PROGRAM _3000_PRG_Running
VAR_IN_OUT
    CurrentStep : ActiveStep;  // Shared step structure with state machine
	NextStep: DINT; // Next step to be modified by sequences
END_VAR
VAR_INPUT
    StepTimerSeconds : DINT;   // Timer value from state machine
    RetrySignal : BOOL;        // Retry signal from state machine
    StateMachineStatus : ST_SM_Status;  // Complete state machine status
END_VAR

VAR
    // Step function blocks for running sequence
    fbStep3000 : FB_SequenceStep;  // Production Start
    fbStep3002 : FB_SequenceStep;  // Production Execute
    fbStep3004 : FB_SequenceStep;  // Production Quality Check
    fbStep3006 : FB_SequenceStep;  // Packaging Prepare
    fbStep3008 : FB_SequenceStep;  // Production Finalize
    
    // Step permissives (simulation for testing)
    step3000Perms : INT := -1;     // All OK for step 3000
    step3002Perms : INT := -1;     // All OK for step 3002
    step3004Perms : INT := -1;     // All OK for step 3004
    step3006Perms : INT := -1;     // All OK for step 3006
    step3008Perms : INT := -1;     // All OK for step 3008
    
END_VAR

//=============================================================================
// PRG_Running - Handles RUNNING state sequence (3000-3999)
//=============================================================================
// Step numbering: 3000, 3002 (even numbers)
// Fault steps: 3001, 3003 (odd numbers, +1 of original)
// NOTE: Initial step setting (CurrentStep.Step = 0) is handled in MAIN program


//=============================================================================
// STEP 3000 - PRODUCTION START
//=============================================================================
fbStep3000(
    inpStep := CurrentStep.Step,
    cfgStep := 3000,
    cfgNextStep := 3002,
    inpStepTimerSeconds := StepTimerSeconds,
    inpRetry := RetrySignal,
    inpStepPermissives := step3000Perms,
    cfgStepTimeout := 12,  // 12 second timeout
    inpFaultStep := FALSE,
    ActiveStep := CurrentStep
);

// Step 3000 Active Logic
IF fbStep3000.outStepActive THEN
    // Only simulate permissives if step is active but not advancing
    IF fbStep3000.outNextStep = fbStep3000.cfgStep THEN  // Step is waiting for permissives
        // Permissives simulation - Simulate based on timer
        IF StepTimerSeconds < 5 THEN
            step3000Perms := 16#FFFE;  // Bit 0 not OK (not ready yet)
        ELSE
            step3000Perms := -1;  // All permissives OK after 5 seconds
        END_IF;
    END_IF;
    
    // HMI configuration and actions
    CurrentStep.PermsHMI.Name := 'Production Start';
    CurrentStep.PermsHMI.Desc[0] := 'Raw Material Available';
    CurrentStep.PermsHMI.Desc[1] := 'Process Temperature OK';
    CurrentStep.PermsHMI.Desc[2] := 'Quality System Ready';
    
    // Add any step-specific actions here
    // Example: Start production line, initialize process parameters, etc.
    
    // FB_SequenceStep determines next step automatically based on permissives
    NextStep := fbStep3000.outNextStep;
ELSE
    // Reset permissives when step is not active (ensures fresh start next time)
    step3000Perms := 16#FFFE;  // Reset to NOT OK when leaving step
END_IF;

//=============================================================================
// STEP 3002 - PRODUCTION EXECUTE
//=============================================================================
fbStep3002(
    inpStep := CurrentStep.Step,
    cfgStep := 3002,
    cfgNextStep := 3004,
    inpStepTimerSeconds := StepTimerSeconds,
    inpRetry := RetrySignal,
    inpStepPermissives := step3002Perms,
    cfgStepTimeout := 20,  // 20 second timeout
    inpFaultStep := FALSE,
    ActiveStep := CurrentStep
);

// Step 3002 Active Logic
IF fbStep3002.outStepActive THEN
    // Only simulate permissives if step is active but not advancing
    IF fbStep3002.outNextStep = fbStep3002.cfgStep THEN  // Step is waiting for permissives
        // Permissives simulation - Simulate based on timer
        IF StepTimerSeconds < 15 THEN
            step3002Perms := 16#FFFD;  // Bit 1 not OK (production not complete)
        ELSE
            step3002Perms := -1;  // All permissives OK after 15 seconds
        END_IF;
    END_IF;
    
    // HMI configuration and actions
    CurrentStep.PermsHMI.Name := 'Production Execute';
    CurrentStep.PermsHMI.Desc[0] := 'Production Line Running';
    CurrentStep.PermsHMI.Desc[1] := 'Quality Checks Passing';
    CurrentStep.PermsHMI.Desc[2] := 'Output Quality OK';
    
    // Add any step-specific actions here
    // Example: Monitor production process, quality checks, output control, etc.
    
    // FB_SequenceStep determines next step automatically based on permissives
    NextStep := fbStep3002.outNextStep;
ELSE
    // Reset permissives when step is not active (ensures fresh start next time)
    step3002Perms := 16#FFFD;  // Reset to NOT OK when leaving step
END_IF;

//=============================================================================
// STEP 3004 - PRODUCTION QUALITY CHECK
//=============================================================================
fbStep3004(
    inpStep := CurrentStep.Step,
    cfgStep := 3004,
    cfgNextStep := 3006,
    inpStepTimerSeconds := StepTimerSeconds,
    inpRetry := RetrySignal,
    inpStepPermissives := step3004Perms,
    cfgStepTimeout := 12,  // 12 second timeout
    inpFaultStep := FALSE,
    ActiveStep := CurrentStep
);

IF fbStep3004.outStepActive THEN
    // Only simulate permissives if step is active but not advancing
    IF fbStep3004.outNextStep = fbStep3004.cfgStep THEN  // Step is waiting for permissives
        // Simulate based on timer: delay bit 2
        IF StepTimerSeconds < 4 THEN
            step3004Perms := 16#FFFB;  // Bit 2 not OK
        ELSE
            step3004Perms := -1;       // All OK
        END_IF;
    END_IF;

    // HMI configuration and actions
    CurrentStep.PermsHMI.Name := 'Production Quality Check';
    CurrentStep.PermsHMI.Desc[0] := 'Inspection Running';
    CurrentStep.PermsHMI.Desc[1] := 'Reject Bin Clear';
    CurrentStep.PermsHMI.Desc[2] := 'Measurements In Spec';

    // Advance handled by FB
    NextStep := fbStep3004.outNextStep;
ELSE
    step3004Perms := 16#FFFB;  // Reset to NOT OK when leaving step
END_IF;

//=============================================================================
// STEP 3006 - PACKAGING PREPARE
//=============================================================================
fbStep3006(
    inpStep := CurrentStep.Step,
    cfgStep := 3006,
    cfgNextStep := 3008,
    inpStepTimerSeconds := StepTimerSeconds,
    inpRetry := RetrySignal,
    inpStepPermissives := step3006Perms,
    cfgStepTimeout := 15,  // 15 second timeout
    inpFaultStep := FALSE,
    ActiveStep := CurrentStep
);

IF fbStep3006.outStepActive THEN
    // Only simulate permissives if step is active but not advancing
    IF fbStep3006.outNextStep = fbStep3006.cfgStep THEN  // Step is waiting for permissives
        // Simulate based on timer: delay bit 3
        IF StepTimerSeconds < 6 THEN
            step3006Perms := 16#FFF7;  // Bit 3 not OK
        ELSE
            step3006Perms := -1;       // All OK
        END_IF;
    END_IF;

    // HMI configuration and actions
    CurrentStep.PermsHMI.Name := 'Packaging Prepare';
    CurrentStep.PermsHMI.Desc[0] := 'Empty Boxes Available';
    CurrentStep.PermsHMI.Desc[1] := 'Labeler Ready';
    CurrentStep.PermsHMI.Desc[2] := 'Conveyor Clear';

    // Advance handled by FB
    NextStep := fbStep3006.outNextStep;
ELSE
    step3006Perms := 16#FFF7;  // Reset to NOT OK when leaving step
END_IF;

//=============================================================================
// STEP 3008 - PRODUCTION FINALIZE
//=============================================================================
fbStep3008(
    inpStep := CurrentStep.Step,
    cfgStep := 3008,
    cfgNextStep := 0,  // sequence complete
    inpStepTimerSeconds := StepTimerSeconds,
    inpRetry := RetrySignal,
    inpStepPermissives := step3008Perms,
    cfgStepTimeout := 10,  // 10 second timeout
    inpFaultStep := FALSE,
    ActiveStep := CurrentStep
);

IF fbStep3008.outStepActive THEN
    // Only simulate permissives if step is active but not advancing
    IF fbStep3008.outNextStep = fbStep3008.cfgStep THEN  // Step is waiting for permissives
        // Simulate based on timer: delay bit 4
        IF StepTimerSeconds < 5 THEN
            step3008Perms := 16#FFEF;  // Bit 4 not OK
        ELSE
            step3008Perms := -1;       // All OK
        END_IF;
    END_IF;

    // HMI configuration and actions
    CurrentStep.PermsHMI.Name := 'Production Finalize';
    CurrentStep.PermsHMI.Desc[0] := 'Batch Closed';
    CurrentStep.PermsHMI.Desc[1] := 'Reports Generated';
    CurrentStep.PermsHMI.Desc[2] := 'Area Clear';

    // Advance handled by FB
    NextStep := fbStep3008.outNextStep;
ELSE
    step3008Perms := 16#FFEF;  // Reset to NOT OK when leaving step
END_IF;

END_PROGRAM

(* stored: Version 1.1.0.1, ProductVersion 3.1.4024.13
   POU _3000_PRG_Running: Id {12345678-1234-1234-1234-123456789002}, SpecialFunc None *)
